FUNCTION_BLOCK GearLever (* Basic FB with empty ECC *)
  (* Standard: 61499-2 *)
  (* Version 1.0, 2021-12-09, Fan *)
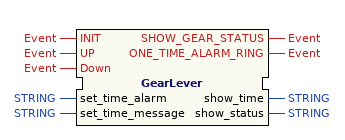
  EVENT_INPUT
    INIT; (* Initialise the Up and Down message at the event *)
    UP; (* Event Up message tick  when pilot press the button *)
    Down; (* Down up message tick when pilot press the button *)
  END_EVENT
  EVENT_OUTPUT
    SHOW_GEAR_STATUS; (* Event to signal that the status has changed *)
    ONE_TIME_ALARM_RING; (* Event to signal that the time alarm is ringing *)
  END_EVENT
  VAR_INPUT
    set_time_alarm : STRING; (* Static input paramter to set the alarm *)
    set_time_message : STRING; (* Static input paramter to set the time in num *)
  END_VAR
  VAR_OUTPUT
    show_time : STRING; (* Show one_time message on pilot input. *)
    show_status : STRING; (* Show gear status *)
  END_VAR
  EC_STATES
    START; (* Initial State *)
  END_STATES
END_FUNCTION_BLOCK
